FUNCTION_BLOCK EL1114
VAR
	_io : EL1xx4_Data;
	{attribute addProperty Name "WcState"}
	_wcState : WcStateInputToggle;
	{attribute addProperty Name "Info data"}
	_infoData : InfoDataBase;
END_VAR

PROPERTY IO : REFERENCE TO EL1xx4_Data
GET
IO REF= _io;
END_GET
END_PROPERTY

PROPERTY WcState : REFERENCE TO WcStateInputToggle
GET
WcState REF= _wcState;
END_GET
END_PROPERTY

END_FUNCTION_BLOCK

(* stored: Version 1.1.0.1, ProductVersion 3.1.4024.9
   POU EL1114: Id {bc43339b-aaeb-0b30-1b9b-c62e6801ed1f}, SpecialFunc None
   Property IO: Id {f7a112ae-6d65-005d-209c-386f21d9a300}
   Get Get: Id {d746fcd2-12b5-04c2-269b-316176e52d78}
   Property WcState: Id {a3e54a06-b60c-0d38-2506-2a46901d80ae}
   Get Get: Id {37a6e02b-5295-08e0-3987-5cdfdd45a35d} *)
